% RSLogix 500 project TWO-CONVEYOR SEQUENCING WITH DELAYED START STOP AND FAULT HANDLING.RSS, saved by version 8.30.00.16 %
PROJECT "PROJ2"    % processor: Bul.1763 MicroLogix 1100 Series B %

PROGRAM FILES
  LAD 2 "MAIN"  4 rungs
  LAD 3 "CONTROLS"  6 rungs
  LAD 4 "IO"  4 rungs
  LAD 5 "ALARMS"  7 rungs

DATA FILES
  O0 OUTPUT  5 elements
  I1 INPUT  14 elements
  S2 STATUS  66 elements
  B3 BINARY  1 elements
  T4 TIMER  2 elements
  C5 COUNTER  1 elements
  R6 CONTROL  1 elements
  N7 INTEGER  1 elements
  F8 FLOAT  1 elements

LADDER 2 "MAIN"
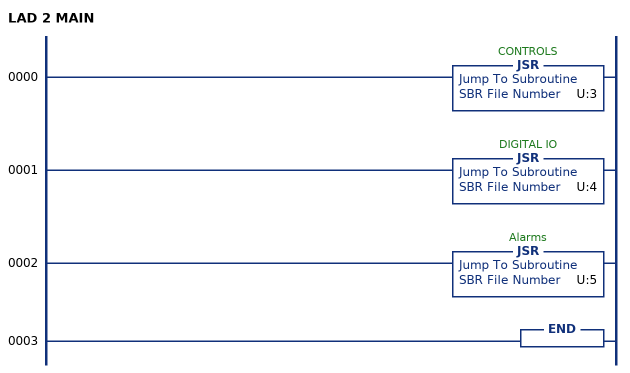
% Rung: 0 %
SOR JSR U:3 EOR
%   U:3  "CONTROLS" %
% Rung: 1 %  % edit flag set %
SOR JSR U:4 EOR
%   U:4  "DIGITAL IO" %
% Rung: 2 %  % edit flag set %
SOR JSR U:5 EOR
%   U:5  "Alarms" %
% Rung: 3 %
SOR END EOR

LADDER 3 "CONTROLS"
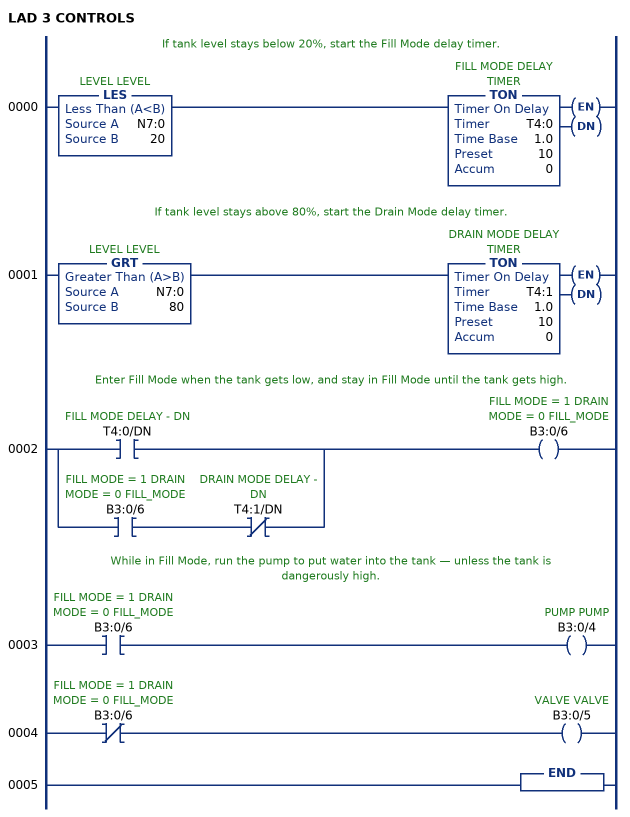
% Rung: 0 %  % edit flag set %
% If tank level stays below 20%, start the Fill Mode delay timer. %
SOR LES N7:0 20 TON T4:0 1.0 10 0 EOR
%   N7:0  LEVEL  "LEVEL" %
%   T4:0  "FILL MODE DELAY TIMER" %
% Rung: 1 %  % edit flag set %
% If tank level stays above 80%, start the Drain Mode delay timer. %
SOR GRT N7:0 80 TON T4:1 1.0 10 0 EOR
%   N7:0  LEVEL  "LEVEL" %
%   T4:1  "DRAIN MODE DELAY TIMER" %
% Rung: 2 %
% Enter Fill Mode when the tank gets low, and stay in Fill Mode until the tank gets high. %
SOR BST XIC T4:0/DN NXB XIC B3:0/6 XIO T4:1/DN BND OTE B3:0/6 EOR
%   T4:0/DN  "FILL MODE DELAY - DN" %
%   B3:0/6  FILL_MODE  "FILL MODE = 1 DRAIN MODE = 0" %
%   T4:1/DN  "DRAIN MODE DELAY - DN" %
% Rung: 3 %
% While in Fill Mode, run the pump to put water into the tank — unless the tank is dangerously high. %
SOR XIC B3:0/6 OTE B3:0/4 EOR
%   B3:0/6  FILL_MODE  "FILL MODE = 1 DRAIN MODE = 0" %
%   B3:0/4  PUMP  "PUMP" %
% Rung: 4 %
SOR XIO B3:0/6 OTE B3:0/5 EOR
%   B3:0/6  FILL_MODE  "FILL MODE = 1 DRAIN MODE = 0" %
%   B3:0/5  VALVE  "VALVE" %
% Rung: 5 %
SOR END EOR

LADDER 4 "IO"
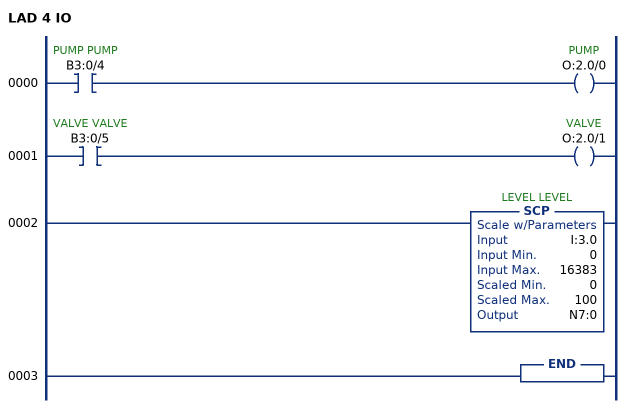
% Rung: 0 %
SOR XIC B3:0/4 OTE O:2.0/0 EOR
%   B3:0/4  PUMP  "PUMP" %
%   O:2.0/0  "PUMP" %
% Rung: 1 %  % edit flag set %
SOR XIC B3:0/5 OTE O:2.0/1 EOR
%   B3:0/5  VALVE  "VALVE" %
%   O:2.0/1  "VALVE" %
% Rung: 2 %  % edit flag set %
SOR SCP I:3.0 0 16383 0 100 N7:0 EOR
%   I:3.0  "LEVEL SENSOR INPUT" %
%   N7:0  LEVEL  "LEVEL" %
% Rung: 3 %
SOR END EOR

LADDER 5 "ALARMS"
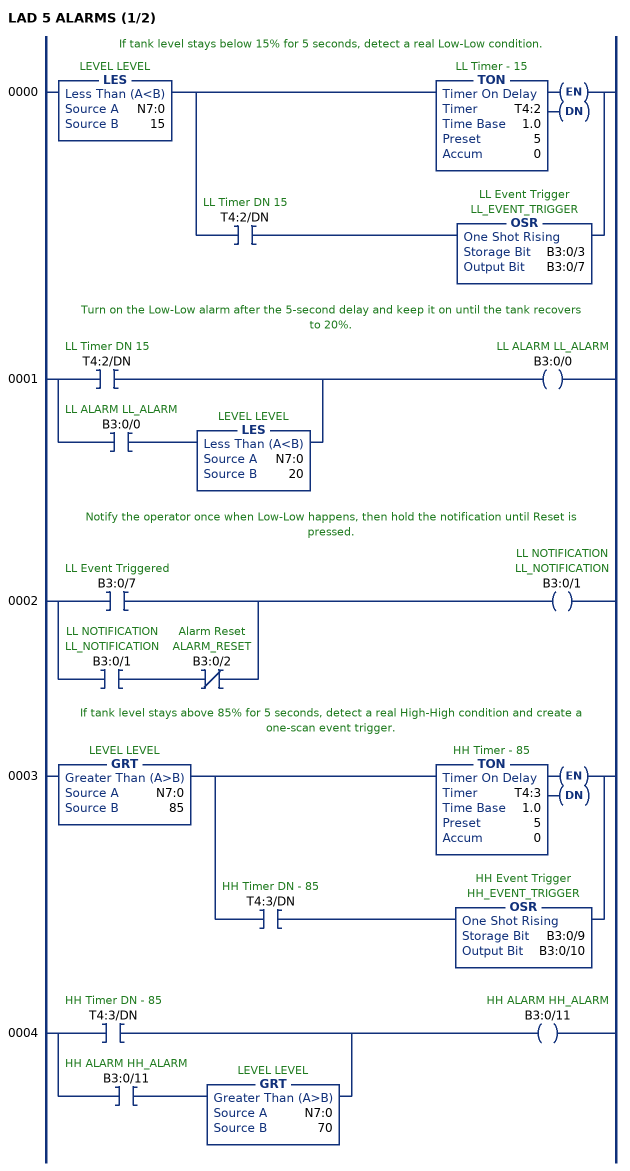
% Rung: 0 %  % edit flag set %
% If tank level stays below 15% for 5 seconds, detect a real Low-Low condition. %
SOR LES N7:0 15 BST TON T4:2 1.0 5 0 NXB XIC T4:2/DN OSR B3:0/3 B3:0/7 BND EOR
%   N7:0  LEVEL  "LEVEL" %
%   T4:2  "LL Timer - 15" %
%   T4:2/DN  "LL Timer DN 15" %
%   B3:0/3  LL_EVENT_TRIGGER  "LL Event Trigger" %
%   B3:0/7  "LL Event Triggered" %
% Rung: 1 %  % edit flag set %
% Turn on the Low-Low alarm after the 5-second delay and keep it on until the tank recovers to 20%. %
SOR BST XIC T4:2/DN NXB XIC B3:0/0 LES N7:0 20 BND OTE B3:0/0 EOR
%   T4:2/DN  "LL Timer DN 15" %
%   B3:0/0  LL_ALARM  "LL ALARM" %
%   N7:0  LEVEL  "LEVEL" %
% Rung: 2 %  % edit flag set %
% Notify the operator once when Low-Low happens, then hold the notification until Reset is pressed. %
SOR BST XIC B3:0/7 NXB XIC B3:0/1 XIO B3:0/2 BND OTE B3:0/1 EOR
%   B3:0/7  "LL Event Triggered" %
%   B3:0/1  LL_NOTIFICATION  "LL NOTIFICATION" %
%   B3:0/2  ALARM_RESET  "Alarm Reset" %
% Rung: 3 %  % edit flag set %
% If tank level stays above 85% for 5 seconds, detect a real High-High condition and create a one-scan event trigger. %
SOR GRT N7:0 85 BST TON T4:3 1.0 5 0 NXB XIC T4:3/DN OSR B3:0/9 B3:0/10 BND EOR
%   N7:0  LEVEL  "LEVEL" %
%   T4:3  "HH Timer - 85" %
%   T4:3/DN  "HH Timer DN - 85" %
%   B3:0/9  HH_EVENT_TRIGGER  "HH Event Trigger" %
%   B3:0/10  HH_EVENT_TRIGGERED  "HH Event Triggered" %
% Rung: 4 %  % edit flag set %
SOR BST XIC T4:3/DN NXB XIC B3:0/11 GRT N7:0 70 BND OTE B3:0/11 EOR
%   T4:3/DN  "HH Timer DN - 85" %
%   B3:0/11  HH_ALARM  "HH ALARM" %
%   N7:0  LEVEL  "LEVEL" %

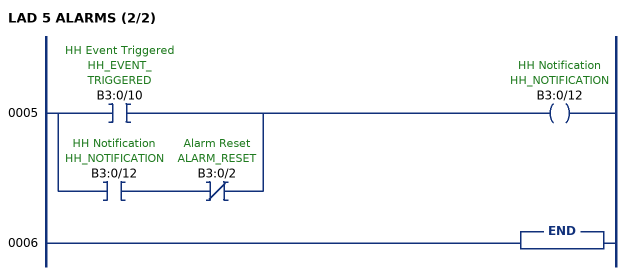
% Rung: 5 %  % edit flag set %
SOR BST XIC B3:0/10 NXB XIC B3:0/12 XIO B3:0/2 BND OTE B3:0/12 EOR
%   B3:0/10  HH_EVENT_TRIGGERED  "HH Event Triggered" %
%   B3:0/12  HH_NOTIFICATION  "HH Notification" %
%   B3:0/2  ALARM_RESET  "Alarm Reset" %
% Rung: 6 %
SOR END EOR

OTHER DOCUMENTED ADDRESSES
  I:0.0/0  "LL SWITCH"
  I:0.0/1  "L SWITCH"
  I:0.0/2  "HH SWITCH"
  I:0.0/3  "H SWITCH"
  N7:1  "HH LEVEL"
  O:0.0/0  "PUMP"

REVISION NOTES
  0: Added alarm sequence

DATA TABLE (non-zero values as saved)
DATA T4
% .PRE .ACC %
% T4:0 % 10 0
% T4:1 % 10 0
